// TIA Portal V17 export
// export: Created 2024-06-14T09:53:12.6922211Z, ExportSetting WithDefaults, DisplayName Totally Integrated Automation Portal, DisplayVersion V17, DisplayName TIA Portal Openness, DisplayVersion V17, DisplayName TIA Portal Version Control Interface, DisplayVersion V17, DisplayName Simotion SCOUT TIA, DisplayVersion 5.4.3.0, DisplayName SINAMICS Startdrive Advanced, DisplayVersion V17 SP1 Update 1, DisplayName SINAMICS Startdrive G110M, G120, G120C, G120D, G120P, G115D, DisplayVersion V17 SP1 Update 1, DisplayName SINAMICS Startdrive G130, G150, S120, S150, SINAMICS MV, S210, DisplayVersion V17 SP1 Update 1, DisplayName STEP 7 Professional, DisplayVersion V17, DisplayName STEP 7 Safety, DisplayVersion V17, DisplayName WinCC Professional, DisplayVersion V17
FUNCTION_BLOCK "CORRECTION_scale_LPG"   // FB11, LAD
{ S7_Optimized_Access := 'TRUE' }
VERSION : 0.1
// stored: AutoNumber false, IsIECCheckEnabled false, IsRetainMemResEnabled false, MemoryReserve 100, SetENOAutomatically false, UDAEnableTagReadback false
   VAR_INPUT
      Stopper_sesnor : Bool;
      Cylinder_presence : Bool;
      Anti_jammer : Bool;
      Start_cycle : Bool;
      Reset_Cycle : Bool;
      Result : Int;
      all_fill_done : Bool;
   END_VAR
   VAR_OUTPUT
      Stopper : Bool;
      LiftTable : Bool;
      Start_correction_Scale : Bool;
      Divider : Bool;
   END_VAR
   VAR
      Check_Scale_Started : Bool;
      Lift_Table { S7_SetPoint := 'True'} : TON_TIME;
      PASS : Bool;
      FAIL : Bool;
      LIFT_down { S7_SetPoint := 'True'} : TON_TIME;
      checking { S7_SetPoint := 'True'} : TON_TIME;
      idx7 : Int;
      p_trig : Array[0..10] of Bool;
   END_VAR
   VAR RETAIN
      Stopper_count { S7_SetPoint := 'True'} : CTU_INT;
   END_VAR
   VAR
      counter_reset : Bool;
      datasend : Bool;
      Filling_done : Bool;
   END_VAR
   VAR_TEMP
      temp : Int;
   END_VAR
   VAR_TEMP   // added for the SCL form of the ladder/FBD networks
      _w1 : Bool;
      _w2 : Bool;
      _w3 : Bool;
   END_VAR
BEGIN

REGION Network 1
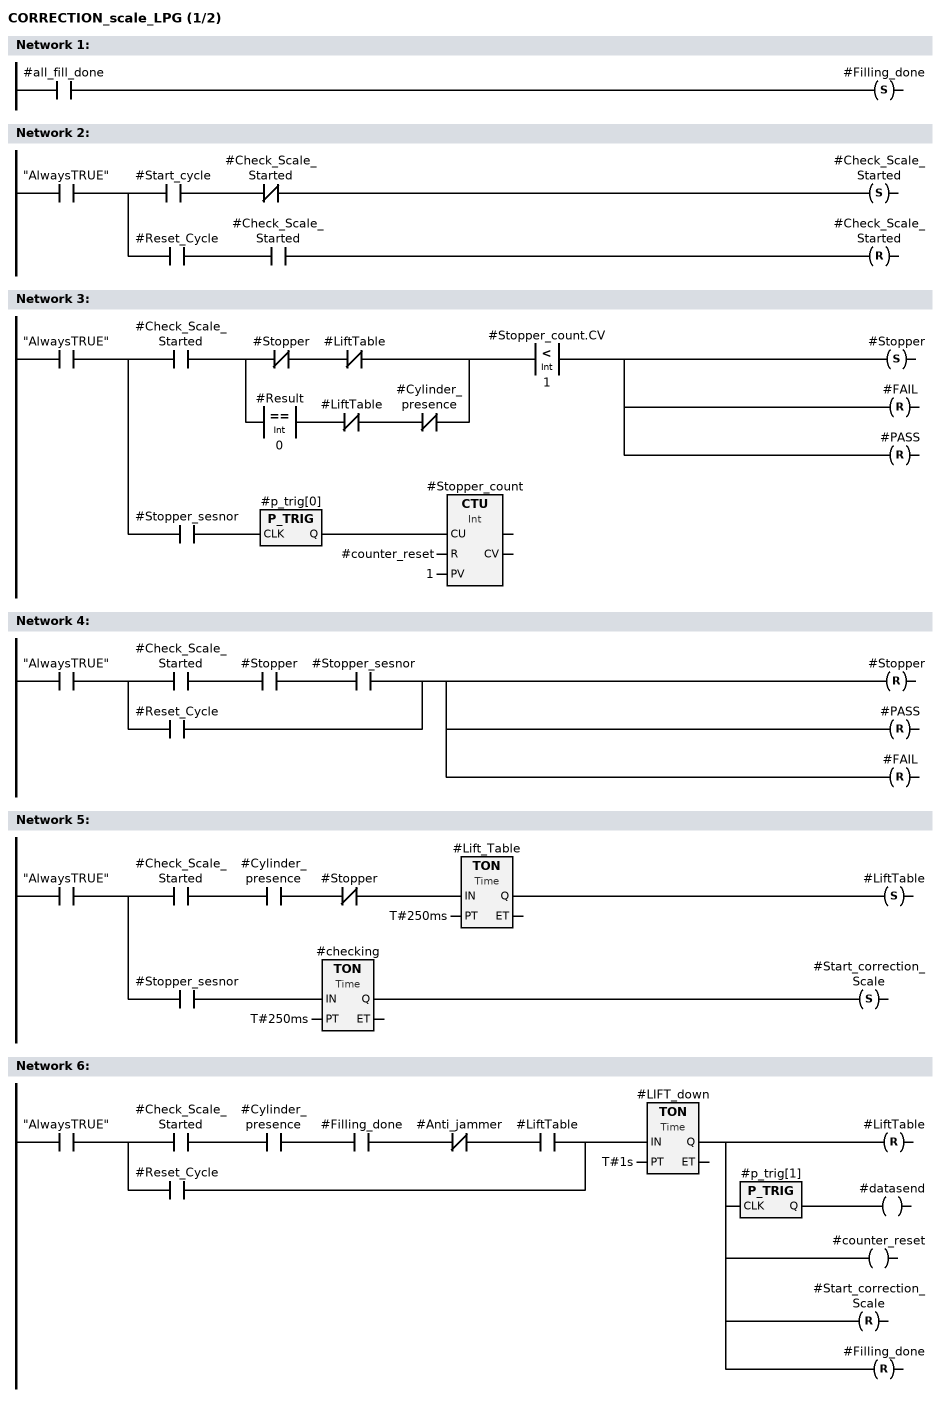
   RUNG wire#powerrail
      Contact( #all_fill_done )
      S_Coil( #Filling_done )
   END_RUNG
   // the same network as SCL:
   IF #all_fill_done THEN #Filling_done := TRUE; END_IF;
END_REGION

REGION Network 2
   RUNG wire#powerrail
      Contact( "AlwaysTRUE" )
      wire#w1
      Contact( #Start_cycle )
      I_Contact( #Check_Scale_Started )
      S_Coil( #Check_Scale_Started )
   END_RUNG
   RUNG wire#w1
      Contact( #Reset_Cycle )
      Contact( #Check_Scale_Started )
      R_Coil( #Check_Scale_Started )
   END_RUNG
   // the same network as SCL:
   IF "AlwaysTRUE" AND #Start_cycle AND NOT #Check_Scale_Started THEN #Check_Scale_Started := TRUE; END_IF;
   IF "AlwaysTRUE" AND #Reset_Cycle AND #Check_Scale_Started THEN #Check_Scale_Started := FALSE; END_IF;
END_REGION

REGION Network 3
   RUNG wire#powerrail
      Contact( "AlwaysTRUE" )
      wire#w1
      Contact( #Check_Scale_Started )
      wire#w2
      I_Contact( #Stopper )
      I_Contact( #LiftTable )
      wire#w3
      { S7_Templates := "SrcType := Int" } LT_Contact(in1 := #Stopper_count.CV, in2 := 1)
      wire#w4
      S_Coil( #Stopper )
   END_RUNG
   RUNG wire#w2
      { S7_Templates := "SrcType := Int" } EQ_Contact(in1 := #Result, in2 := 0)
      I_Contact( #LiftTable )
      I_Contact( #Cylinder_presence )
   END_RUNG wire#w3
   RUNG wire#w4
      R_Coil( #FAIL )
   END_RUNG
   RUNG wire#w4
      R_Coil( #PASS )
   END_RUNG
   RUNG wire#w1
      Contact( #Stopper_sesnor )
      P_Trig( #p_trig[0] )
      { S7_Templates := "value_type := Int" } #Stopper_count.CTU(r := #counter_reset, pv := 1, cv =>)
   END_RUNG
   // the same network as SCL:
   #_w1 := "AlwaysTRUE" AND #Check_Scale_Started AND ((NOT #Stopper AND NOT #LiftTable) OR ((#Result = 0) AND NOT #LiftTable AND NOT #Cylinder_presence)) AND (#Stopper_count.CV < 1);
   IF #_w1 THEN
       #Stopper := TRUE;
       #FAIL := FALSE;
       #PASS := FALSE;
   END_IF;
   #_w2 := "AlwaysTRUE" AND #Stopper_sesnor;
   #_w3 := #_w2 AND NOT #p_trig[0];   // rising edge
   #p_trig[0] := #_w2;
   #Stopper_count(CU := #_w3, R := #counter_reset, PV := 1);   // CTU
END_REGION

REGION Network 4
   RUNG wire#powerrail
      Contact( "AlwaysTRUE" )
      wire#w1
      Contact( #Check_Scale_Started )
      Contact( #Stopper )
      Contact( #Stopper_sesnor )
      wire#w2
      R_Coil( #Stopper )
   END_RUNG
   RUNG wire#w1
      Contact( #Reset_Cycle )
   END_RUNG wire#w2
   RUNG wire#w2
      R_Coil( #PASS )
   END_RUNG
   RUNG wire#w2
      R_Coil( #FAIL )
   END_RUNG
   // the same network as SCL:
   #_w1 := "AlwaysTRUE" AND ((#Check_Scale_Started AND #Stopper AND #Stopper_sesnor) OR #Reset_Cycle);
   IF #_w1 THEN
       #Stopper := FALSE;
       #PASS := FALSE;
       #FAIL := FALSE;
   END_IF;
END_REGION

REGION Network 5
   RUNG wire#powerrail
      Contact( "AlwaysTRUE" )
      wire#w1
      Contact( #Check_Scale_Started )
      Contact( #Cylinder_presence )
      I_Contact( #Stopper )
      { S7_Templates := "time_type := Time" } #Lift_Table.TON(pt := T#250ms, et =>)
      S_Coil( #LiftTable )
   END_RUNG
   RUNG wire#w1
      Contact( #Stopper_sesnor )
      { S7_Templates := "time_type := Time" } #checking.TON(pt := T#250ms, et =>)
      S_Coil( #Start_correction_Scale )
   END_RUNG
   // the same network as SCL:
   #Lift_Table(IN := "AlwaysTRUE" AND #Check_Scale_Started AND #Cylinder_presence AND NOT #Stopper,   // TON
               PT := T#250ms);
   IF #Lift_Table.Q THEN #LiftTable := TRUE; END_IF;
   #checking(IN := "AlwaysTRUE" AND #Stopper_sesnor, PT := T#250ms);   // TON
   IF #checking.Q THEN #Start_correction_Scale := TRUE; END_IF;
END_REGION

REGION Network 6
   RUNG wire#powerrail
      Contact( "AlwaysTRUE" )
      wire#w1
      Contact( #Check_Scale_Started )
      Contact( #Cylinder_presence )
      Contact( #Filling_done )
      I_Contact( #Anti_jammer )
      Contact( #LiftTable )
      wire#w2
      { S7_Templates := "time_type := Time" } #LIFT_down.TON(pt := T#1s, et =>)
      wire#w3
      R_Coil( #LiftTable )
   END_RUNG
   RUNG wire#w1
      Contact( #Reset_Cycle )
   END_RUNG wire#w2
   RUNG wire#w3
      P_Trig( #p_trig[1] )
      Coil( #datasend )
   END_RUNG
   RUNG wire#w3
      Coil( #counter_reset )
   END_RUNG
   RUNG wire#w3
      R_Coil( #Start_correction_Scale )
   END_RUNG
   RUNG wire#w3
      R_Coil( #Filling_done )
   END_RUNG
   // the same network as SCL:
   #LIFT_down(IN := "AlwaysTRUE" AND ((#Check_Scale_Started AND #Cylinder_presence AND #Filling_done AND NOT #Anti_jammer AND #LiftTable) OR #Reset_Cycle),   // TON
              PT := T#1s);
   IF #LIFT_down.Q THEN #LiftTable := FALSE; END_IF;
   #_w1 := #LIFT_down.Q AND NOT #p_trig[1];   // rising edge
   #p_trig[1] := #LIFT_down.Q;
   #datasend := #_w1;
   #counter_reset := #LIFT_down.Q;
   IF #LIFT_down.Q THEN
       #Start_correction_Scale := FALSE;
       #Filling_done := FALSE;
   END_IF;
END_REGION

REGION Network 7
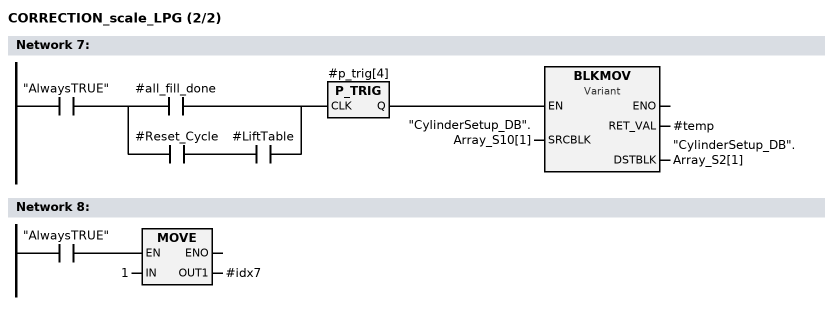
   RUNG wire#powerrail
      Contact( "AlwaysTRUE" )
      wire#w1
      Contact( #all_fill_done )
      wire#w2
      P_Trig( #p_trig[4] )
      { S7_Templates := "blk_type := Variant" } BLKMOV(SRCBLK := "CylinderSetup_DB".Array_S10[1], RET_VAL => #temp, DSTBLK => "CylinderSetup_DB".Array_S2[1])
   END_RUNG
   RUNG wire#w1
      Contact( #Reset_Cycle )
      Contact( #LiftTable )
   END_RUNG wire#w2
   // the same network as SCL:
   #_w1 := "AlwaysTRUE" AND (#all_fill_done OR (#Reset_Cycle AND #LiftTable));
   #_w2 := #_w1 AND NOT #p_trig[4];   // rising edge
   #p_trig[4] := #_w1;
   IF #_w2 THEN
       #temp := BLKMOV(SRCBLK := "CylinderSetup_DB".Array_S10[1], DSTBLK => "CylinderSetup_DB".Array_S2[1]);
   END_IF;
END_REGION

REGION Network 8
   RUNG wire#powerrail
      Contact( "AlwaysTRUE" )
      Move(in := 1, out1 => #idx7)
   END_RUNG
   // the same network as SCL:
   IF "AlwaysTRUE" THEN #idx7 := 1; END_IF;
END_REGION
END_FUNCTION_BLOCK
